(* IEC 61131-3 sources: plcassist-cli/packages/volt-lsp-iec/test-corpus/awa-palletizer/Device/Plc Logic/Application/999 Library NextGen 01/999.002 Standard Objects, 13 files *)

(* ---- libCylinder.fb ---- *)
{attribute 'symbol' := 'none'}
FUNCTION_BLOCK libCylinder EXTENDS libModuleHandler
VAR_IN_OUT
	// Interface to HMI
	_HMI: dutHMI;
END_VAR
VAR_INPUT
	// Automatic out
	xCmdGoOut : BOOL := FALSE;
	// Automatic in
	xCmdGoIn : BOOL := FALSE;
	// Sensor cylinder is out
	SenOut : libDI;
	// Sensor out travel time before error
	tErrTimeOutSensorOut : TIME := T#0MS;
	// Sensor cylinder is in
	SenIn : libDI;
	// Sensor in travel time before error
	tErrTimeOutSensorIn : TIME := T#0MS;
	// Sensor simulation
	xSensorSimulation: BOOL := FALSE;
	tSimulationTravelTime: TIME := T#0S;
	// Interlock in
	xInterlIn: BOOL := FALSE;
	// Interlock out
	xInterlOut: BOOL := FALSE;
END_VAR
VAR_OUTPUT
	// Cylinder is out
	xCylIsOut : BOOL := FALSE;
	// Cylinder is in
	xCylIsIn : BOOL := FALSE;
	// Move the Cylinder out
	xGoOut: BOOL := FALSE;
	// Move the Cylinder in
	xGoIn: BOOL := FALSE;
END_VAR
VAR
	// Timer on delay
	fbTravelTimeIn : TON;
	// Timer on delay
	fbTravelTimeOut: TON;
	// Timer simulation
	fbSimulationIn: TON;
	// Timer simulation
	fbSimulationOut: TON;
	// Sensor simulation
	xSimGoOut: BOOL := FALSE;
	// Sendor simulation
	xSimGoIn: BOOL := FALSE;

	//Alarm
	xErrTimeOut_GoOut : BOOL := FALSE;
	// Alarm
	xErrTimeOut_GoIn : BOOL := FALSE;
	// Condition out
	xOutAllowed: BOOL := FALSE;
	// Condition in
	xInAllowed: BOOL := FALSE;
	// Interlock causes no output
	xInterlocked: BOOL := FALSE;
END_VAR

//------------------------------------------------------------------------------------------
// This function controls a Cylinder object.
//
// 11-04-2022 RPo Initial version.
//
//------------------------------------------------------------------------------------------

// ### LOGIC ###
{region}
	IF (xInit) THEN
		xInit             	:= FALSE;

		_HMI.strName 		:= strName;
		_HMI.wCmd 			:= 0;
		_HMI.wStatus 		:= 0;

		_HMI.wCmd.0 		:= TRUE;	// 0 = Manual, 1 = Auto
		_HMI.wCmd.1			:= FALSE; 	// Out.
		_HMI.wCmd.2			:= FALSE;	// In.

		xExecute		 	:= TRUE;
		xCmdReset			:= FALSE;

		xGoIn				:= FALSE;
		xGoOut				:= FALSE;

		xInterlIn			:= FALSE;
		xInterlOut			:= FALSE;

		xErrTimeOut_GoOut 	:= FALSE;
		xErrTimeOut_GoIn  	:= FALSE;

		myClassType       	:= enClassType.ctCylinder;
	END_IF

	//
	// Reset manual control after estop.
	//
	IF (xCmdEStopActive) THEN
		_HMI.wCmd.1			:= FALSE; 	// Forward.
		_HMI.wCmd.2			:= FALSE;	// Reverse.
	END_IF

	//
	// Determine if output is allowed, without interlock.
	//
	xOutAllowed := ((    _HMI.wCmd.0 AND xExecute AND xCmdGoOut  AND NOT xCmdGoIn ) OR
					(NOT _HMI.wCmd.0 AND _HMI.wCmd.1 AND NOT _HMI.wCmd.2 ))
				   AND NOT xErrTimeOut_GoOut AND NOT xErrTimeOut_GoIn;

	xInAllowed  := ((    _HMI.wCmd.0 AND xExecute AND xCmdGoIn   AND NOT xCmdGoOut) OR
					(NOT _HMI.wCmd.0 AND _HMI.wCmd.2  AND NOT _HMI.wCmd.1 ))
				   AND NOT xErrTimeOut_GoOut AND NOT xErrTimeOut_GoIn;

	//
	// Determine if the output is interlocked for display status.
	//
	xInterlocked := (xOutAllowed AND xInterlOut) OR (xInAllowed  AND xInterlIn);

	//
	// Interlock the output if necessary....
	//
	xOutAllowed := xOutAllowed AND NOT xInterlOut;
	xInAllowed  := xInAllowed  AND NOT xInterlIn;

	xGoOut := xOutAllowed;
	xGoIn  := xInAllowed;

	// Remember the status of the cylinder in simulation mode. Or use
	// use direct inputs in non-simulation. For cylinders with no input
	// sensors this may be valuable. This only works for bi-stable
	// cylinders.

	IF (xSensorSimulation) THEN
		xSimGoOut S= xGoOut;
		xSimGoOut R= xGoIn;

		xSimGoIn  S= xGoIn;
		xSimGoIn  R= xGoOut;

		fbSimulationIn( IN := xSimGoIn, PT := tSimulationTravelTime);
		fbSimulationOut(IN := xSimGoOut, PT := tSimulationTravelTime);

		xCylIsIn := fbSimulationIn.Q;
		xCylIsOut := fbSimulationOut.Q;
	ELSE
		xCylIsIn  := SenIn.xDI;
		xCylIsOut := SenOut.xDI;
	END_IF

	// Monitor the cylinder movement.

	IF (tErrTimeOutSensorIn > T#0S) THEN
		fbTravelTimeIn (IN := (xGoIn  AND NOT xCylIsIn ), PT := tErrTimeOutSensorIn );
	END_IF

	IF (tErrTimeOutSensorOut > T#0S) THEN
		fbTravelTimeOut(IN := (xGoOut AND NOT xCylIsOut), PT := tErrTimeOutSensorOut);
	END_IF
{endregion}

// ### ALARM ###
{region}
	//ERROR: Timeout
	xErrTimeOut_GoIn  := xErrTimeOut_GoIn  OR fbTravelTimeIn.Q;
	xErrTimeOut_GoOut := xErrTimeOut_GoOut OR fbTravelTimeOut.Q;

	IF (xCmdReset) THEN
		xErrTimeOut_GoOut 	  := FALSE;
		xErrTimeOut_GoIn  	  := FALSE;
	END_IF
{endregion}

// ### ERROR  ###
{region}
	xCMError := xCMError OR xErrTimeOut_GoOut OR xErrTimeOut_GoIn;
{endregion}

// ### VISUAL ###
{region}
	//Alarm
	_HMI.wStatus.0 := _HMI.wCmd.0;			// Automatic
	_HMI.wStatus.1 := NOT(_HMI.wCmd.0);		// Manual
	_HMI.wStatus.2 := xErrTimeOut_GoOut;
	_HMI.wStatus.3 := xErrTimeOut_GoIn;
	_HMI.wStatus.4 := xErrTimeOut_GoOut OR xErrTimeOut_GoIn;
	_HMI.wStatus.5 := xInterlOut;
	_HMI.wStatus.6 := xInterlIn;
	_HMI.wStatus.7 := xInterlocked;
	_HMI.wStatus.8 := xGoOut;
	_HMI.wStatus.9 := xGoIn;
	_HMI.wStatus.10 := xGoOut OR xGoIn;
{endregion}

{region}
	//------------------------------------------------------------------------------------------------------
	// Alarm and warning handling.
	//------------------------------------------------------------------------------------------------------

	wErrorID := 16#0000;
	wWarningID := 16#0000;

	IF (xErrTimeOut_GoOut) THEN wErrorID := 16#0004; END_IF
	IF (xErrTimeOut_GoIn) THEN wWarningID := 16#0005; END_IF

	//Alarm
	ALM_Error(
		ModuleHandler:= myModuleHandler,
		ErrorHandler:= ,
		xSetError:= (wErrorID <> 0),
		eSeverity:= L_IE1P.L_IE1P_SeverityLevel.Fault,
		wTextRefId:= lib_TextList,
		wErrorId:= wErrorID,
		eReaction:= L_IE1P.L_IE1P_Reaction.NormalStop);

	//Warning
	ALM_Warning(
		ModuleHandler:= myModuleHandler,
		ErrorHandler:= ,
		xSetError:= (wWarningID <> 0),
		eSeverity:= L_IE1P.L_IE1P_SeverityLevel.Warning,
		wTextRefId:= lib_TextList,
		wErrorId:= wWarningID,
		eReaction:= L_IE1P.L_IE1P_Reaction.No_Reaction);

	IF NOT xInitProgramAlarms THEN
		myModuleHandler.SetParent(ModuleHandlerParent:= IQ_ModuleHandler);
		xInitProgramAlarms:= TRUE;
	END_IF

	ForwardAlarms(
		xEnable:= TRUE,
		ModuleHandler:= myModuleHandler,
		xForwardFromChildModules:=TRUE);
{endregion}

END_FUNCTION_BLOCK

(* ---- libDI.fb ---- *)
{attribute 'symbol' := 'none'}
FUNCTION_BLOCK libDI EXTENDS libObject
VAR_IN_OUT
	// Interface to HMI
	_HMI: dutHMI;
END_VAR

VAR_INPUT
	// Sensor value
	xInput : BOOL := FALSE;
	// On delay
	tOnDelay : TIME := T#0MS;
	// Off delay
	tOffDelay : TIME := T#0MS;

END_VAR
VAR_OUTPUT
	// Sensor output value
	xDI : BOOL := FALSE;
	// Sensor rising trigger
	xDIeu : BOOL := FALSE;
	// Sensor falling trigger
	xDIed : BOOL := FALSE;
END_VAR
VAR
	// On delay
	TON_Delay : TON;
	// Off delay
	TOF_Delay : TOF;
	// Rising trigger
	RTRIG_euX : R_TRIG;
	// Falling trigger
	FTRIG_edX : F_TRIG;
END_VAR

//------------------------------------------------------------------------------------------
// This function controls a digital input.
//------------------------------------------------------------------------------------------

// ### LOGIC ###
{region}
	IF (xInit) THEN
		xInit             	:= FALSE;

		_HMI.strName 		:= strName;
		_HMI.wCmd 			:= 0;
		_HMI.wStatus 		:= 0;

		_HMI.wCmd.0 		:= TRUE;	// 0 = Manual, 1 = Auto
		_HMI.wCmd.1			:= FALSE; 	// Value.

		myClassType 		:= enClassType.ctDI;
	END_IF

	IF (_HMI.wCmd.0) THEN
		IF (xInput) THEN
			TON_Delay(IN := TRUE, PT := tOnDelay);
			xDI := TON_Delay.Q;
			TOF_Delay(IN := xDI);
		ELSE
			TOF_Delay(IN := FALSE, PT := tOffDelay);
			xDI := TOF_Delay.Q;
			TON_Delay(IN := xDI);
		END_IF
	ELSE
		xDI := _HMI.wCmd.1;
	END_IF

	RTRIG_euX(CLK := xDI, Q => xDIeu);
	FTRIG_edX(CLK := xDI, Q => xDIed);
{endregion}

// ### ALARM ###
{region}

{endregion}

// ### VISUAL ###
{region}
	_HMI.wStatus.0 := _HMI.wCmd.0;			// Automatic
	_HMI.wStatus.1 := NOT(_HMI.wCmd.0);		// Manual
	_HMI.wStatus.2 := xDI;
{endregion}

END_FUNCTION_BLOCK

(* ---- libDO.fb ---- *)
{attribute 'symbol' := 'none'}
FUNCTION_BLOCK libDO EXTENDS libObject
VAR_IN_OUT
	// Interface to HMI
	_HMI: dutHMI;
END_VAR

VAR_INPUT
	// Output value
	xDO : BOOL := FALSE;
	// On delay
	tOnDelay : TIME := T#0MS;
	// Off delay
	tOffDelay : TIME := T#0MS;

	// Interlock causes no output
	xInterlocked: BOOL := FALSE;
END_VAR
VAR_OUTPUT
	// Output value
	xOutput : BOOL := FALSE;
	// Rising edge
	xDOeu : BOOL := FALSE;
	// Falling edge
	xDOed : BOOL := FALSE;
END_VAR
VAR
	// On delay
	TON_Delay : TON;
	// Off delay
	TOF_Delay : TOF;
	// Rising edge
	RTRIG_euX : R_TRIG;
	// Falling edge
	FTRIG_edX : F_TRIG;
END_VAR

//------------------------------------------------------------------------------------------
// This function controls a digital output.
//
// 11-04-2022 RPo Initial version.
//
//------------------------------------------------------------------------------------------

// ### LOGIC ###
{region}
	IF (xInit) THEN
		xInit       		:= FALSE;

		_HMI.strName 		:= strName;
		_HMI.wCmd			:= 0;
		_HMI.wCmd.0 		:= TRUE;	// 0 = Manual, 1 = Auto
		_HMI.wCmd.1			:= FALSE; 	// On/Off.
		_HMI.wCmd.2			:= FALSE;	// Blink.
		_HMI.wStatus		:= 0;

		xExecute		 	:= TRUE;
		xCmdReset			:= FALSE;
		xDO					:= FALSE;

 		xInterlocked 		:= FALSE;

		myClassType			:= enClassType.ctDO;
	END_IF

	IF (_HMI.wCmd.0) THEN
		IF (xDO) THEN
			TOF_Delay(IN := TRUE);
			TON_Delay(IN := TRUE, PT := tOnDelay);
			xOutput := TON_Delay.Q;
		ELSE
			TON_Delay(IN := FALSE);
			TOF_Delay(IN := FALSE, PT := tOffDelay);
			xOutput := TOF_Delay.Q;
		END_IF
	END_IF

	IF (NOT _HMI.wCmd.0) THEN
		xOutput := _HMI.wCmd.1;
	END_IF;

	xOutput := xOutput AND NOT xInterlocked;

	RTRIG_euX(CLK := xOutput, Q => xDOeu);
	FTRIG_edX(CLK := xOutput, Q => xDOed);
{endregion}

// ### ALARM ###
{region}

{endregion}

// ### VISUAL ###
{region}
	_HMI.wStatus.0 := _HMI.wCmd.0;			// Automatic
	_HMI.wStatus.1 := NOT(_HMI.wCmd.0);		// Manual
	_HMI.wStatus.2 := xInterlocked;
	_HMI.wStatus.3 := xDO;
{endregion}

END_FUNCTION_BLOCK

(* ---- libInverter.fb ---- *)
FUNCTION_BLOCK libInverter EXTENDS libModuleHandler
VAR_IN_OUT
	// Interface to HMI
	_HMI: dutHMI;
END_VAR
VAR_INPUT
	// Automatic forward
	xCmdGoForw : BOOL := FALSE;
	// Automatic backward
	xCmdGoBackw : BOOL := FALSE;
	// Setpoint
	rSetpoint: REAL := 0;
	// Switch delay from direction
	tSwitchDelay : TIME := T#100MS;
	// Interlock forward
	xInterlForw : BOOL := FALSE;
	// Interlock backward
	xInterlBackw : BOOL := FALSE;
	//Alarm
	xThermFault : BOOL := FALSE;
END_VAR
VAR_OUTPUT
	// Output forward
	xOutForw : BOOL := FALSE;
	// Output backward
	xOutBackw : BOOL := FALSE;
END_VAR
VAR_INPUT
	// Start next timer
	tStartNext : TIME := T#1S;
	// Stop next timer
	tStopNext: TIME := T#1S;
END_VAR
VAR_OUTPUT
	// Start next allowed.
	xStartNext : BOOL;
	// Stop next allowed.
	xStopNext: BOOL;
	// At stand still velocity
	xStandstillVelocity: BOOL;
END_VAR
VAR
	// Timer switch direction
	fbSwitchOk : TON;
	// Switch direction allowed
	xSwitchOk : BOOL := FALSE;
	// Falling trigger forward output
	fbFTrigForw : F_TRIG;
	// Falling trigger backward output
	fbFTrigBackw : F_TRIG;
	// Timer start next allowed.
	fbStartNext : TON;
	// Timer stop next allowed.
	fbStopNext: TOF;

	//Alarm
	xErrThermFault : BOOL := FALSE;
	// Condition forward
	xForwAllowed: BOOL := FALSE;
	// Condition backward
	xBackwAllowed: BOOL := FALSE;
	// Interlock causes no output
	xInterlocked: BOOL := FALSE;
	// Visual output
	byModeVisual: BYTE := 0;

	eTB2PAxisErrorId: L_TB2P.L_IE1P_Error;

	// Short access to errors
	eAxisErrorId: WORD;
END_VAR
VAR_INPUT
		// Motion state Inverter
	TB2P_Inverter: L_TB2P_BasicMotionBase;
END_VAR

VAR_IN_OUT
	// Inverter Axis
	AxisRef: AXIS_REF;
END_VAR
VAR
	iState: INT;
END_VAR

// ### LOGIC ###
{region}
	IF (xInit) THEN
		xInit            	:= FALSE;

		_HMI.strName 		:= strName;
		_HMI.wCmd 			:= 0;
		_HMI.wCmd.0 		:= TRUE;	// 0 = Manual, 1 = Auto
		_HMI.wCmd.1			:= FALSE; 	// Forward.
		_HMI.wCmd.2			:= FALSE;	// Reverse.
		_HMI.wStatus		:= 0;

		xExecute		 	:= TRUE;
		xCmdReset			:= FALSE;
		xCmdGoBackw	  	 	:= FALSE;
		xCmdGoForw		 	:= FALSE;

		xInterlForw			:= FALSE;
		xInterlBackw		:= FALSE;

		xErrThermFault   	:= FALSE;

		myClassType      	:= enClassType.ctMotor;
	END_IF

	//
	// Reset manual control after estop.
	//
	IF (xCmdEStopActive) THEN
		_HMI.wCmd.1			:= FALSE; 	// Forward.
		_HMI.wCmd.2			:= FALSE;	// Reverse.
	END_IF

	//
	// Determine if output is allowed, without interlock.
	//
	xForwAllowed  := ( (    _HMI.wCmd.0 AND xExecute AND xCmdGoForw  AND NOT xCmdGoBackw) OR
					   (NOT _HMI.wCmd.0 AND _HMI.wCmd.1 AND NOT _HMI.wCmd.2))
					 AND NOT xErrThermFault AND NOT xCmdEStopActive AND xSwitchOk;

	xBackwAllowed := ( (    _HMI.wCmd.0 AND xExecute AND xCmdGoBackw AND NOT xCmdGoForw ) OR
					   (NOT _HMI.wCmd.0 AND _HMI.wCmd.2 AND NOT _HMI.wCmd.1 ))
					 AND NOT xErrThermFault AND NOT xCmdEStopActive AND xSwitchOk;

	//
	// Determine if the output is interlocked for display status.
	//
	xInterlocked  := (xForwAllowed  AND xInterlForw) OR (xBackwAllowed AND xInterlBackw);

	//
	// Interlock the output if necessary....
	//
	xForwAllowed  := xForwAllowed  AND NOT xInterlForw  AND NOT xCmdEStopActive;
	xBackwAllowed := xBackwAllowed AND NOT xInterlBackw AND NOT xCmdEStopActive;

	//
	//Switch direction ok
	//

	fbSwitchOk(IN := NOT xOutForw AND NOT xOutBackw, PT := tSwitchDelay);

	IF (fbSwitchOk.Q) THEN
		xSwitchOk := TRUE;
	END_IF

	fbFTrigForw(CLK  := xOutForw );
	fbFTrigBackw(CLK := xOutBackw);

	IF (fbFTrigForw.Q OR fbFTrigBackw.Q) THEN
		xSwitchOk := FALSE;
	END_IF

	//Output
	xOutForw  := xForwAllowed;
	xOutBackw := xBackwAllowed;

	// Start next
	fbStartNext(IN := (TB2P_Inverter.lrActVel > 1.0), PT := tStartNext);
	xStartNext := fbStartNext.Q;

	// Stop next
	fbStopNext(IN := xOutForw, PT := tStopNext);
	xStopNext := fbStopNext.Q;

	IF (eTB2PAxisErrorId <> L_TB2P.L_IE1P_Error.NoError) THEN
		TB2P_Inverter.xResetError := NOT TB2P_Inverter.xResetError AND xCmdReset;
		iState := 0;
	END_IF

	CASE iState OF
	0: 	TB2P_Inverter.xEnable := (eTB2PAxisErrorId = L_TB2P.L_IE1P_Error.NoError);
		TB2P_Inverter.xEnableOperation := FALSE;

		TB2P_Inverter.xQSPApplication := TRUE;
		TB2P_Inverter.scCtrlBasicMotion.xMoveVelExecute := FALSE;
		TB2P_Inverter.xAbort := FALSE;

		IF (TB2P_Inverter.xReadyForOperation AND TB2P_Inverter.xEnable)  THEN
			TB2P_Inverter.xResetError := FALSE;
			iState := 2;
		END_IF

	2:  TB2P_Inverter.xEnableOperation := FALSE;
		TB2P_Inverter.xQSPApplication := TRUE;
		TB2P_Inverter.scCtrlBasicMotion.xMoveVelExecute := FALSE;

		IF xOutForw THEN // Check enable operation.
			TB2P_Inverter.xEnableOperation := TRUE;

			IF (TB2P_Inverter.xReadyForMotion) THEN
				TB2P_Inverter.xResetError := FALSE;
				iState := 10;
			END_IF
		END_IF

	10:	TB2P_Inverter.xQSPApplication := FALSE;
		TB2P_Inverter.scPar.eDirection := MC_DIRECTION.mcPositiveDirection;
		TB2P_Inverter.scPar.lrVel      := rSetpoint;
		TB2P_Inverter.scCtrlBasicMotion.xMoveVelExecute := TRUE;
		TB2P_Inverter.scPar.lrAcc		:= 500;
		TB2P_Inverter.scPar.lrDec		:= 500;
		TB2P_Inverter.scPar.lrJerk      := 0;

		IF NOT xOutForw THEN
			iState := 20;
		END_IF

	20: TB2P_Inverter.scCtrlBasicMotion.xMoveVelExecute := FALSE;
		TB2P_Inverter.xAbort := TRUE;
		TB2P_Inverter.scPar.lrVel  := 0.0;

		IF NOT TB2P_Inverter.scStatusBasicMotion.xFunDone THEN
			iState := 30;
		END_IF

	30: IF TB2P_Inverter.scStatusBasicMotion.xFunDone THEN
			TB2P_Inverter.xAbort := FALSE;
			iState := 0;
		END_IF

	END_CASE

	TB2P_Inverter(  xEnable := TRUE,
	     		    Axis := AxisRef);

	eAxisErrorId    := AxisRef.eActiveErrorID;
	eTB2PAxisErrorId:= TB2P_Inverter.eErrorID;

	IF (AxisRef.xSTOActive) THEN
		eAxisErrorId    := 0;
		eTB2PAxisErrorId:= 0;
		iState := 0;
	END_IF

	xStandstillVelocity := TB2P_Inverter.scStatusBasicMotion.xStandstillActVelocity;

// ### ALARM ###
{region}
	IF (xCmdReset) THEN
		xErrThermFault := FALSE;
	END_IF

	xErrThermFault := (xThermFault OR xErrThermFault OR (eTB2PAxisErrorId <> L_TB2P.L_IE1P_Error.NoError));
{endregion}

// ### ERROR  ###
{region}
	xCMError := xCMError OR xErrThermFault;
{endregion}

// ### VISUAL ###
{region}
	//Alarm
	_HMI.wStatus.0 := _HMI.wCmd.0;				// Automatic
	_HMI.wStatus.1 := NOT(_HMI.wCmd.0);			// Manual
	_HMI.wStatus.2 := xErrThermFault;			// Fault
	_HMI.wStatus.3 := xInterlForw;				// Interlock forward
	_HMI.wStatus.4 := xInterlBackw;				// Interlock backward
	_HMI.wStatus.5 := xInterlocked;				// Interlocked
	_HMI.wStatus.6 := xOutForw;					// Output forward
	_HMI.wStatus.7 := xOutBackw;				// Output backward
	_HMI.wStatus.8 := xOutForw OR xOutBackw;	// Output
{endregion}

{region}
	//------------------------------------------------------------------------------------------------------
	// Alarm and warning handling.
	//------------------------------------------------------------------------------------------------------

	wErrorID := 16#0000;
	wWarningID := 16#0000;

	IF (xThermFault) THEN wErrorID := 16#0001; END_IF
	IF (xInterlForw) THEN wWarningID := 16#0002; END_IF
	IF (xInterlBackw) THEN wWarningID := 16#0003; END_IF

	//Alarm
	ALM_Error(
		ModuleHandler:= myModuleHandler,
		ErrorHandler:= ,
		xSetError:= (wErrorID <> 0),
		eSeverity:= L_IE1P.L_IE1P_SeverityLevel.Fault,
		wTextRefId:= lib_TextList,
		wErrorId:= wErrorID,
		eReaction:= L_IE1P.L_IE1P_Reaction.NormalStop);

	//Warning
	ALM_Warning(
		ModuleHandler:= myModuleHandler,
		ErrorHandler:= ,
		xSetError:= (wWarningID <> 0),
		eSeverity:= L_IE1P.L_IE1P_SeverityLevel.Warning,
		wTextRefId:= lib_TextList,
		wErrorId:= wWarningID,
		eReaction:= L_IE1P.L_IE1P_Reaction.No_Reaction);

	IF NOT xInitProgramAlarms THEN
		myModuleHandler.SetParent(ModuleHandlerParent:= IQ_ModuleHandler);
		AxisRef.ModuleHandler.SetParent(ModuleHandlerParent := IQ_ModuleHandler);

		xInitProgramAlarms:= TRUE;
	END_IF

	ForwardAlarms(
		xEnable:= TRUE,
		ModuleHandler:= myModuleHandler,
		xForwardFromChildModules:=TRUE);
{endregion}

END_FUNCTION_BLOCK

(* ---- libModuleHandler.fb ---- *)
{attribute 'symbol' := 'none'}
FUNCTION_BLOCK ABSTRACT libModuleHandler EXTENDS libObject

VAR_IN_OUT
	// Parent handler
	IQ_ModuleHandler : L_IMHP_ModuleHandler;
END_VAR

VAR
	// my handler
	myModuleHandler : L_IMHP_ModuleHandler;
	// Connect alarms to parent
	xInitProgramAlarms: BOOL := FALSE;
	// Error ID
	wErrorID: UINT := 0;
	// Warning ID
	wWarningID: UINT := 0;
	// Forward alarms
	ForwardAlarms : L_IE1P_ForwardSeverity;
	// Warning
	ALM_Warning : L_IE1P_SetErrorSingle;
	// Error
	ALM_Error : L_IE1P_SetErrorSingle;
END_VAR

//------------------------------------------------------------------------------------------
// General object definition.
//
// 11-04-2022 RPo Initial version.
//
//------------------------------------------------------------------------------------------

END_FUNCTION_BLOCK

(* ---- libMotor.fb ---- *)
{attribute 'symbol' := 'none'}
FUNCTION_BLOCK libMotor EXTENDS libModuleHandler
VAR_IN_OUT
	// Interface to HMI
	_HMI: dutHMI;
END_VAR
VAR_INPUT
	// Automatic forward
	xCmdGoForw : BOOL := FALSE;
	// Automatic backward
	xCmdGoBackw : BOOL := FALSE;
	// Switch delay from direction
	tSwitchDelay : TIME := T#100MS;
	// Interlock forward
	xInterlForw : BOOL := FALSE;
	// Interlock backward
	xInterlBackw : BOOL := FALSE;
	//Alarm
	xThermFault : BOOL := FALSE;
	// Start next timer
	tStartNext : TIME := T#1S;
	// Stop next timer
	tStopNext: TIME := T#1S;
END_VAR
VAR_OUTPUT
	// Output forward
	xOutForw : BOOL := FALSE;
	// Output backward
	xOutBackw : BOOL := FALSE;
	// Start next allowed.
	xStartNext : BOOL;
	// Stop next allowed.
	xStopNext: BOOL;
END_VAR
VAR
	// Timer switch direction
	fbSwitchOk : TON;
	// Switch direction allowed
	xSwitchOk : BOOL := FALSE;
	// Falling trigger forward output
	fbFTrigForw : F_TRIG;
	// Falling trigger backward output
	fbFTrigBackw : F_TRIG;
	// Timer start next allowed.
	fbStartNext : TON;
	// Timer stop next allowed.
	fbStopNext: TOF;

	//Alarm
	xErrThermFault : BOOL := FALSE;
	// Condition forward
	xForwAllowed: BOOL := FALSE;
	// Condition backward
	xBackwAllowed: BOOL := FALSE;
	// Interlock causes no output
	xInterlocked: BOOL := FALSE;
END_VAR

//------------------------------------------------------------------------------------------
// This function controls a motor object.
//------------------------------------------------------------------------------------------

// ### LOGIC ###
{region}
	IF (xInit) THEN
		xInit            	:= FALSE;

		_HMI.strName 		:= strName;
		_HMI.wCmd			:= 0;
		_HMI.wCmd.0 		:= TRUE;	// 0 = Manual, 1 = Auto
		_HMI.wCmd.1			:= FALSE; 	// Forward.
		_HMI.wCmd.2			:= FALSE;	// Reverse.
		_HMI.wStatus		:= 0;

		xExecute		 	:= TRUE;
		xCmdReset			:= FALSE;
		xCmdGoBackw	  	 	:= FALSE;
		xCmdGoForw		 	:= FALSE;

		xInterlForw			:= FALSE;
		xInterlBackw		:= FALSE;

		xErrThermFault   	:= FALSE;

		myClassType      	:= enClassType.ctMotor;
	END_IF

	//
	// Reset manual control after estop.
	//
	IF (xCmdEStopActive) THEN
		_HMI.wCmd.1			:= FALSE; 	// Forward.
		_HMI.wCmd.2			:= FALSE;	// Reverse.
	END_IF

	//
	// Determine if output is allowed, without interlock.
	//
	xForwAllowed  := ( (    _HMI.wCmd.0 AND xExecute AND xCmdGoForw  AND NOT xCmdGoBackw) OR
					   (NOT _HMI.wCmd.0 AND _HMI.wCmd.1 AND NOT _HMI.wCmd.2))
					 AND NOT xErrThermFault AND NOT xCmdEStopActive AND xSwitchOk;

	xBackwAllowed := ( (    _HMI.wCmd.0 AND xExecute AND xCmdGoBackw AND NOT xCmdGoForw ) OR
					   (NOT _HMI.wCmd.0 AND _HMI.wCmd.2 AND NOT _HMI.wCmd.1 ))
					 AND NOT xErrThermFault AND NOT xCmdEStopActive AND xSwitchOk;

	//
	// Determine if the output is interlocked for display status.
	//
	xInterlocked  := (xForwAllowed  AND xInterlForw) OR (xBackwAllowed AND xInterlBackw);

	//
	// Interlock the output if necessary....
	//
	xForwAllowed  := xForwAllowed  AND NOT xInterlForw  AND NOT xCmdEStopActive;
	xBackwAllowed := xBackwAllowed AND NOT xInterlBackw AND NOT xCmdEStopActive;

	//
	//Switch direction ok
	//

	fbSwitchOk(IN := NOT xOutForw AND NOT xOutBackw, PT := tSwitchDelay);

	IF (fbSwitchOk.Q) THEN
		xSwitchOk := TRUE;
	END_IF

	fbFTrigForw(CLK  := xOutForw );
	fbFTrigBackw(CLK := xOutBackw);

	IF (fbFTrigForw.Q OR fbFTrigBackw.Q) THEN
		xSwitchOk := FALSE;
	END_IF

	//Output
	xOutForw  := xForwAllowed;
	xOutBackw := xBackwAllowed;

	// Start next
	fbStartNext(IN := xOutForw, PT := tStartNext);
	xStartNext := fbStartNext.Q;

	// Stop next
	fbStopNext(IN := xOutForw, PT := tStopNext);
	xStopNext := fbStopNext.Q;

{endregion}

// ### ALARM ###
{region}
	IF (xCmdEStopActive) THEN
		//
		// In case of an emergency stop the termical fault can be ignored...
		//
		xThermFault    := FALSE;
		xErrThermFault := FALSE;
	END_IF

	IF (xCmdReset) THEN
		xErrThermFault 		  := FALSE;
	END_IF

	xErrThermFault := (xThermFault OR xErrThermFault);
{endregion}

// ### ERROR  ###
{region}
	xCMError := xCMError OR xErrThermFault;
{endregion}

// ### VISUAL ###
{region}
	_HMI.wStatus.0 := _HMI.wCmd.0;			// Automatic
	_HMI.wStatus.1 := NOT(_HMI.wCmd.0);		// Manual
	_HMI.wStatus.2 := xErrThermFault;
	_HMI.wStatus.3 := xInterlForw;
	_HMI.wStatus.4 := xInterlBackw;
	_HMI.wStatus.5 := xInterlocked;
	_HMI.wStatus.6 := xOutForw;
	_HMI.wStatus.7 := xOutBackw;
	_HMI.wStatus.8 := xOutForw OR xOutBackw;
{endregion}

{region}
	//------------------------------------------------------------------------------------------------------
	// Alarm and warning handling.
	//------------------------------------------------------------------------------------------------------

	wErrorID := 16#0000;
	wWarningID := 16#0000;

	IF (xThermFault) THEN wErrorID := 16#0001; END_IF
	IF (xInterlForw) THEN wWarningID := 16#0002; END_IF
	IF (xInterlBackw) THEN wWarningID := 16#0003; END_IF

	//Alarm
	ALM_Error(
		ModuleHandler:= myModuleHandler,
		ErrorHandler:= ,
		xSetError:= (wErrorID <> 0),
		eSeverity:= L_IE1P.L_IE1P_SeverityLevel.Fault,
		wTextRefId:= lib_TextList,
		wErrorId:= wErrorID,
		eReaction:= L_IE1P.L_IE1P_Reaction.NormalStop);

	//Warning
	ALM_Warning(
		ModuleHandler:= myModuleHandler,
		ErrorHandler:= ,
		xSetError:= (wWarningID <> 0),
		eSeverity:= L_IE1P.L_IE1P_SeverityLevel.Warning,
		wTextRefId:= lib_TextList,
		wErrorId:= wWarningID,
		eReaction:= L_IE1P.L_IE1P_Reaction.No_Reaction);

	IF NOT xInitProgramAlarms THEN
		myModuleHandler.SetParent(ModuleHandlerParent:= IQ_ModuleHandler);
		xInitProgramAlarms:= TRUE;
	END_IF

	ForwardAlarms(
		xEnable:= TRUE,
		ModuleHandler:= myModuleHandler,
		xForwardFromChildModules:=TRUE);
{endregion}

END_FUNCTION_BLOCK

(* ---- libObject.fb ---- *)
{attribute 'symbol' := 'none'}
FUNCTION_BLOCK ABSTRACT libObject
VAR_OUTPUT
	// Error
	xCMError: BOOL;
END_VAR

VAR_INPUT
	// Name of the object
	strName: STRING[30] := 'OBJECT';
	// Execute logic in automatic state
	xExecute: BOOL := TRUE;
	// Reset the error
	xCmdReset: BOOL := FALSE;
	// First time execution
	xInit: BOOL := TRUE;
END_VAR

VAR_OUTPUT
	// What type of class am I
	myClassType: enClassType;;
END_VAR

VAR_INPUT
	// Emergency stop is active
	xCmdEStopActive: BOOL := FALSE;
END_VAR

//------------------------------------------------------------------------------------------
// General object definition.
//
// 11-04-2022 RPo Initial version.
//
//------------------------------------------------------------------------------------------

END_FUNCTION_BLOCK

METHOD isClassType : BOOL
VAR_INPUT
	pClassType: enClassType;
END_VAR
isClassType := (myClassType = pClassType);
END_METHOD

(* ---- libSafetyDI.fb ---- *)
{attribute 'symbol' := 'none'}
FUNCTION_BLOCK libSafetyDI EXTENDS libObject
VAR_IN_OUT
	// Interface to HMI
	_HMI: dutHMI;
END_VAR

VAR_INPUT
	// Sensor value
	xInput : BOOL := FALSE;
	// On delay
	tOnDelay : TIME := T#0MS;
	// Off delay
	tOffDelay : TIME := T#0MS;

END_VAR
VAR_OUTPUT
	// Sensor output value
	xDI : BOOL := FALSE;
	// Sensor rising trigger
	xDIeu : BOOL := FALSE;
	// Sensor falling trigger
	xDIed : BOOL := FALSE;
END_VAR
VAR
	// On delay
	TON_Delay : TON;
	// Off delay
	TOF_Delay : TOF;
	// Rising trigger
	RTRIG_euX : R_TRIG;
	// Falling trigger
	FTRIG_edX : F_TRIG;
END_VAR

//------------------------------------------------------------------------------------------
// This function controls a digital input.
//------------------------------------------------------------------------------------------

// ### LOGIC ###
{region}
	IF (xInit) THEN
		xInit             	:= FALSE;

		_HMI.strName 		:= strName;
		_HMI.wCmd 			:= 0;
		_HMI.wStatus 		:= 0;

		_HMI.wCmd.0 		:= TRUE;	// 0 = Manual, 1 = Auto
		_HMI.wCmd.1			:= FALSE; 	// Value.

		myClassType 		:= enClassType.ctDI;
	END_IF

	IF (_HMI.wCmd.0) THEN
		IF (xInput) THEN
			TON_Delay(IN := TRUE, PT := tOnDelay);
			xDI := TON_Delay.Q;
			TOF_Delay(IN := xDI);
		ELSE
			IF (xCmdReset) THEN
				xDI := FALSE;
			END_IF
		END_IF
	ELSE
		xDI := _HMI.wCmd.1;
	END_IF

	RTRIG_euX(CLK := xDI, Q => xDIeu);
	FTRIG_edX(CLK := xDI, Q => xDIed);
{endregion}

// ### ALARM ###
{region}

{endregion}

// ### VISUAL ###
{region}
	_HMI.wStatus.0 := _HMI.wCmd.0;			// Automatic
	_HMI.wStatus.1 := NOT(_HMI.wCmd.0);		// Manual
	_HMI.wStatus.2 := xDI;
{endregion}

END_FUNCTION_BLOCK

(* ---- libSetpoint.fb ---- *)
{attribute 'symbol' := 'none'}
FUNCTION_BLOCK libSetpoint EXTENDS libModuleHandler
VAR_IN_OUT
	// Interface to HMI
	_HMI: dutSetpointHMI;
END_VAR
VAR_INPUT RETAIN PERSISTENT
	// Scaled setpoint
	rSetpoint_Auto: REAL := 50;
END_VAR
VAR_INPUT
	// Scaled maximum
	rMax: REAL := 100;
	// Scaled high value
	rHi: REAL := 100;
	// Scaled low value
	rLo: REAL := 0;
	// Scaled minimum
	rMin: REAL := 0;
	// Unscaled maximum
	uiAOMax: UINT := 4096;
	// Unscaled minimum
	uiAOMin: UINT := 0;
END_VAR
VAR_OUTPUT
	// Analogue output
	uiAO: UINT := 0;
END_VAR
VAR
	rSetpoint: REAL := 0;
	// Real values to calculate with
	rScale: REAL := 0;
	rAOMax: REAL := 0;
	rAOMin: REAL := 0;
	rAO: REAL := 0;
	// Error
	xSetpointError: BOOL := FALSE;
END_VAR

//------------------------------------------------------------------------------------------
// This function scales a setpoint to analogue output value using a scaling factor.
// The value is also limited to the uiHi and uiLo value. If the value of uiHi or uiLo
// equals 0, the limit is ignored.
//
// 11-04-2022 RPo Initial version.
//
//------------------------------------------------------------------------------------------

// ### LOGIC ###
{region}
	IF (xInit) THEN
		xInit          		:= FALSE;

		_HMI.strName 		:= strName;
		_HMI.wCmd 			:= 0;
		_HMI.wStatus 		:= 0;

		_HMI.wCmd.0 		:= TRUE;	// 0 = Manual, 1 = Auto
		_HMI.rSetpoint_Manual := 30.0;

		xExecute		 	:= TRUE;
		xCmdReset			:= FALSE;

		xSetpointError 		:= FALSE;

		myClassType    		:= enClassType.ctSetpoint;
	END_IF

	// Determine which setpoint to use....
	IF (_HMI.wCmd.0) THEN
		rSetpoint := rSetpoint_Auto;
	ELSE
		rSetpoint := _HMI.rSetpoint_Manual;
	END_IF

	// If not execute, setpoint drops to minimum...
	IF (NOT xExecute) THEN
		rSetpoint := rMin;
	END_IF

	// Limit checks.
	IF (rSetpoint > rMax) THEN
		rSetpoint := rMax;
	END_IF

	IF (rSetpoint < rMin) THEN
		rSetpoint := rMin;
	END_IF

	IF (rSetpoint > rHi) AND (rHi > 0) THEN
		rSetpoint       := rHi;
	END_IF

	IF (rSetpoint < rLo) AND (rLo > 0) THEN
		rSetpoint       := rLo;
	END_IF

	uiAO := uiAOMin;

	IF (rMax - rMin > 0) AND (uiAOMax - uiAOMin >0)  THEN
		rAOMax := UINT_TO_REAL(uiAOMax);
		rAOMin := UINT_TO_REAL(uiAOMin);

		rScale := (rAOMax - rAOMin) / (rMax - rMin);
		rAO := rScale * rSetpoint;

		uiAO := REAL_TO_UINT(rAO);
	ELSE
		xSetpointError := TRUE;
	END_IF
{endregion}

// ### ERROR  ###
{region}
	IF (xCmdReset) THEN
		xSetpointError 		  := FALSE;
	END_IF

	xCMError := xCMError OR xSetpointError;
{endregion}

// ### VISUAL ###
{region}
	_HMI.strName := strName;

	_HMI.wStatus.0 := _HMI.wCmd.0;			// Automatic
	_HMI.wStatus.1 := NOT(_HMI.wCmd.0);		// Manual
	_HMI.wStatus.2 := xSetpointError;
	_HMI.rHi := rHi;
	_HMI.rLo := rLo;
{endregion}

END_FUNCTION_BLOCK

(* ---- libSFCHandler.fb ---- *)
{attribute 'symbol' := 'none'}
FUNCTION_BLOCK ABSTRACT libSFCHandler
VAR_IN_OUT
	// Parent handler
	IQ_ModuleHandler : L_IMHP_ModuleHandler;
END_VAR

VAR
	// my handler
	myModuleHandler : L_IMHP_ModuleHandler;
	// Connect alarms to parent
	xInitProgramAlarms: BOOL := FALSE;
	// Error ID
	wErrorID: UINT := 0;
	// Warning ID
	wWarningID: UINT := 0;
	// Forward alarms
	ForwardAlarms : L_IE1P_ForwardSeverity;
	// Warning
	ALM_Warning : L_IE1P_SetErrorSingle;
	// Error
	ALM_Error : L_IE1P_SetErrorSingle;
END_VAR

//------------------------------------------------------------------------------------------
// General object definition.
//
// 11-04-2022 RPo Initial version.
//
//------------------------------------------------------------------------------------------

END_FUNCTION_BLOCK

(* ---- libSIG.fb ---- *)
{attribute 'symbol' := 'none'}
FUNCTION_BLOCK libSIG EXTENDS libObject
VAR_IN_OUT
	// Interface to HMI
	_HMI: dutHMI;
END_VAR

VAR_INPUT
	// Output value
	xDO : BOOL := FALSE;
	// Blinking
	xDO_Blink: BOOL := FALSE;
	// On delay
	tOnDelay : TIME := T#0MS;
	// Off delay
	tOffDelay : TIME := T#0MS;
	// Blink time high
	tTimeHigh: TIME := T#600MS;
	// Blink time low
	tTimeLow: TIME := T#600MS;

	// Interlock causes no output
	xInterlocked: BOOL := FALSE;
END_VAR
VAR_OUTPUT
	// Output value
	xOutput : BOOL := FALSE;
	// Rising edge
	xDOeu : BOOL := FALSE;
	// Falling edge
	xDOed : BOOL := FALSE;
END_VAR
VAR

	// On delay
	TON_Delay : TON;
	// Off delay
	TOF_Delay : TOF;
	// Rising edge
	RTRIG_euX : R_TRIG;
	// Falling edge
	FTRIG_edX : F_TRIG;
	// Blinking
	Blink: BLINK;
END_VAR

//------------------------------------------------------------------------------------------
// This function controls a signal object.
//
// 11-04-2022 RPo Initial version.
//
//------------------------------------------------------------------------------------------

// ### LOGIC ###
{region}
	IF (xInit) THEN
		xInit       		:= FALSE;

		_HMI.strName 		:= strName;
		_HMI.wCmd			:= 0;
		_HMI.wStatus		:= 0;

		_HMI.wCmd.0 		:= TRUE;	// 0 = Manual, 1 = Auto
		_HMI.wCmd.1			:= FALSE; 	// On/Off.
		_HMI.wCmd.2			:= FALSE;	// Blink.

		xExecute		 	:= TRUE;
		xCmdReset			:= FALSE;

		myClassType 		:= enClassType.ctSIG;
	END_IF

	Blink(ENABLE := TRUE, TIMEHIGH := tTimeHigh, TIMELOW:= tTimeLow);

	IF (_HMI.wCmd.0) THEN
		IF (xDO) THEN
			IF (xDO_Blink) THEN
				xOutput := Blink.OUT;
			ELSE
				TOF_Delay(IN := TRUE);
				TON_Delay(IN := TRUE, PT := tOnDelay);
				xOutput := TON_Delay.Q;
			END_IF;
		END_IF

	ELSE
		xOutput := _HMI.wCmd.1;

		IF _HMI.wCmd.2 THEN
			xOutput := Blink.OUT;
		END_IF
	END_IF;

	xOutput := xOutput AND NOT xInterlocked;

	RTRIG_euX(CLK := xOutput, Q => xDOeu);
	FTRIG_edX(CLK := xOutput, Q => xDOed);
{endregion}

// ### ALARM ###
{region}

{endregion}

// ### VISUAL ###
{region}
	_HMI.wStatus.0 := _HMI.wCmd.0;			// Automatic
	_HMI.wStatus.1 := NOT(_HMI.wCmd.0);		// Manual
	_HMI.wStatus.2 := xInterlocked;
	_HMI.wStatus.3 := xDO;
{endregion}

END_FUNCTION_BLOCK

(* ---- libTimer.fb ---- *)
FUNCTION_BLOCK libTimer
VAR_INPUT
	IN: BOOL;
	PAUSE: BOOL;
	PT: TIME;
END_VAR
VAR_OUTPUT
	Q: BOOL;
	ET: TIME;
END_VAR
VAR
	fbTON: TON;
	fbIN_RT: R_TRIG;
	iState: INT;
	tTime: TIME;
END_VAR

fbIN_RT(CLK := IN);

CASE iState OF
0 : 	fbTON(IN := FALSE, PT := PT);
		Q := FALSE;
		ET := T#0S;

	 	IF (fbIN_RT.Q) THEN
			tTime := PT;
			fbTON(IN := TRUE, PT := tTime);
			Q := TRUE;

	 		iState := 100;
	 	END_IF

100:	fbTON(IN := TRUE, PT := tTime);
		Q := TRUE;
		ET := fbTON.ET;

	 	IF (fbIN_RT.Q) THEN
			fbTON(IN := FALSE, PT := tTime);
		END_IF

		IF (fbTON.Q) THEN
			Q := FALSE;

			iState := 0;
		END_IF

		IF (PAUSE) THEN
			Q := FALSE;

			tTime := fbTON.PT - fbTON.ET;
			fbTON(IN := FALSE, PT := tTime);

			iState := 200;
		END_IF

200:	fbTON(IN := FALSE, PT := tTime);
		Q := FALSE;

		IF NOT(PAUSE) THEN
			iState := 100;
		END_IF
END_CASE

END_FUNCTION_BLOCK

(* ---- libWatchDog.fb ---- *)
{attribute 'symbol' := 'none'}
FUNCTION_BLOCK libWatchDog
VAR_INPUT
	// Counter from the communication
	uiCounter: UINT := 0;
END_VAR
VAR
	// Previous value
	uiPrevCounter: UINT := 0;
END_VAR
VAR_OUTPUT
	// Counter does not change withing TIME
	{attribute 'symbol' := 'read'}
	xError: BOOL := FALSE;
END_VAR
VAR
	// Timer
	TimeOut_TON: TON;
	// Time out time
	TimeOut_TIME: TIME := T#5S;
END_VAR

//------------------------------------------------------------------------------------------
// This function is a watchdog.
//
// 11-04-2022 RPo Initial version.
//
//------------------------------------------------------------------------------------------

// Compare values. If equal start timer.....

TimeOut_TON(IN := (uiCounter = uiPrevCounter), PT := TimeOut_TIME );

// Save for next time...

uiPrevCounter := uiCounter;

// Value does not change withing specified time out....

xError := TimeOut_TON.Q;

END_FUNCTION_BLOCK
